FUNCTION_BLOCK A_Tag IMPLEMENTS Debug.I_Debug

//FB_Init is always available implicitly and it is used primarily for initialization.
//The return value is not evaluated. For a specific influence, you can also declare the
//methods explicitly and provide additional code there with the standard initialization
//code. You can evaluate the return value.
METHOD FB_Init: BOOL
VAR_INPUT
    bInitRetains: BOOL; // TRUE: the retain variables are initialized (reset warm / reset cold)
    bInCopyCode: BOOL;  // TRUE: the instance will be copied to the copy code afterward (online change)
	
	iTag			: I_Tag;
	refTag			: REFERENCE TO I_Tag;
END_VAR
IF NOT __ISVALIDREF(refTag) THEN
	Debug.DebugMsg(THIS^, ': Ref = 0!');
	RETURN;
END_IF

IF iTag = 0 THEN
	Debug.DebugMsg(THIS^, ': Itf = 0!');
	RETURN;
END_IF

IF refTag <> 0 THEN
	Debug.DebugMsg(THIS^, ': Ref itf should be unassigned!');
	RETURN;
END_IF

refTag := iTag;
END_METHOD

END_FUNCTION_BLOCK

(* stored: Version 1.1.0.1
   POU A_Tag: Id {8a40967c-8a31-41b2-94f0-e498695d817c}, SpecialFunc None
   Method FB_Init: Id {d40d420e-518b-45f7-b2db-cc6e8991e8df} *)
